SYSTEM CODEC_TEST2L (* PUBL/SUBL Test with Derived Data Types *)
  (* Standard: 61499-1ITA; Classification: Communications; Function: Test System *)
  (* Version 0.9, 2004-06-23, JHC, Rockwell Automation, Deleted MONITOR (not used). *)
  (* Version 0.8, 2004-06-22, JHC, Rockwell Automation, Modified to use IN_MATRIX, OUT_MATRIX. *)
  (* Version 0.7, 2003-12-04, JHC, Rockwell Automation, Removed QI's from PUBL/SUBLs *)
  (* Version 0.6, 2002-03-08, JHC, Rockwell Automation, Added M_IO for MATRIX I/O *)
  (* Version 0.5, 2002-03-06, JHC, Rockwell Automation, Added TEST_MATRIX, single TEST frame *)
  (* Version 0.4, 2001-06-13, JHC, Rockwell Automation, Added applications including TEST_AI16C. *)
  (* Version 0.3, 2001-06-08, JHC, Rockwell Automation, Corrected UDP addresses; changed GUIs to IN_ANY, OUT_ANY *)
  (* Version 0.2, 2001-05-30, JHC, Rockwell Automation, Saved layouts *)
  (* Version 0.1, 2000-05-16, JHC, Rockwell Automation, File type changed to ".sys" *)
  (* Version 0.0, 2000-04-19, JHC, Rockwell Automation *)
  APPLICATION TEST_REAL_VS
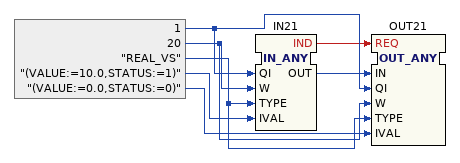
    FBS
      IN21 : IN_ANY;
      OUT21 : OUT_ANY;
    END_FBS
    EVENT_CONNECTIONS
      IN21.IND TO OUT21.REQ;
    END_CONNECTIONS
    DATA_CONNECTIONS
      IN21.OUT TO OUT21.IN;
      1 TO IN21.QI;
      20 TO IN21.W;
      "REAL_VS" TO IN21.TYPE;
      "(VALUE:=10.0,STATUS:=1)" TO IN21.IVAL;
      1 TO OUT21.QI;
      20 TO OUT21.W;
      "REAL_VS" TO OUT21.TYPE;
      "(VALUE:=0.0,STATUS:=0)" TO OUT21.IVAL;
    END_CONNECTIONS
  END_APPLICATION
  APPLICATION TEST_ENUMS
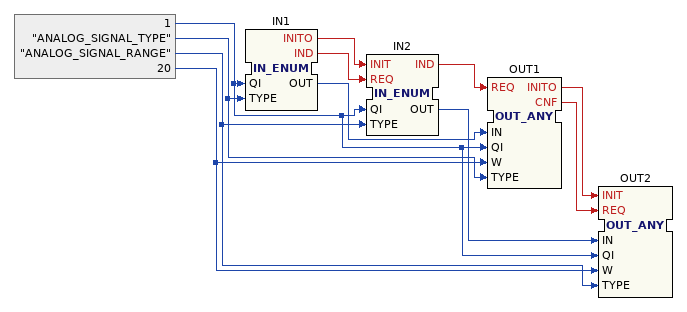
    FBS
      IN1 : IN_ENUM;
      IN2 : IN_ENUM;
      OUT1 : OUT_ANY;
      OUT2 : OUT_ANY;
    END_FBS
    EVENT_CONNECTIONS
      IN1.INITO TO IN2.INIT;
      IN1.IND TO IN2.REQ;
      IN2.IND TO OUT1.REQ;
      OUT1.INITO TO OUT2.INIT;
      OUT1.CNF TO OUT2.REQ;
    END_CONNECTIONS
    DATA_CONNECTIONS
      IN1.OUT TO OUT1.IN;
      IN2.OUT TO OUT2.IN;
      1 TO IN1.QI;
      "ANALOG_SIGNAL_TYPE" TO IN1.TYPE;
      1 TO IN2.QI;
      "ANALOG_SIGNAL_RANGE" TO IN2.TYPE;
      1 TO OUT1.QI;
      20 TO OUT1.W;
      "ANALOG_SIGNAL_TYPE" TO OUT1.TYPE;
      1 TO OUT2.QI;
      20 TO OUT2.W;
      "ANALOG_SIGNAL_RANGE" TO OUT2.TYPE;
    END_CONNECTIONS
  END_APPLICATION
  APPLICATION TEST_FREQ
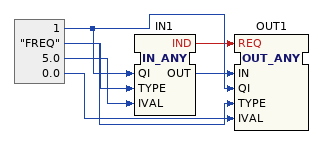
    FBS
      IN1 : IN_ANY;
      OUT1 : OUT_ANY;
    END_FBS
    EVENT_CONNECTIONS
      IN1.IND TO OUT1.REQ;
    END_CONNECTIONS
    DATA_CONNECTIONS
      IN1.OUT TO OUT1.IN;
      1 TO IN1.QI;
      "FREQ" TO IN1.TYPE;
      5.0 TO IN1.IVAL;
      1 TO OUT1.QI;
      "FREQ" TO OUT1.TYPE;
      0.0 TO OUT1.IVAL;
    END_CONNECTIONS
  END_APPLICATION
  APPLICATION TEST_SUBR
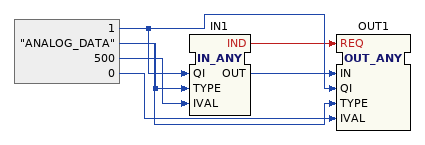
    FBS
      IN1 : IN_ANY;
      OUT1 : OUT_ANY;
    END_FBS
    EVENT_CONNECTIONS
      IN1.IND TO OUT1.REQ;
    END_CONNECTIONS
    DATA_CONNECTIONS
      IN1.OUT TO OUT1.IN;
      1 TO IN1.QI;
      "ANALOG_DATA" TO IN1.TYPE;
      500 TO IN1.IVAL;
      1 TO OUT1.QI;
      "ANALOG_DATA" TO OUT1.TYPE;
      0 TO OUT1.IVAL;
    END_CONNECTIONS
  END_APPLICATION
  APPLICATION TEST_AI16
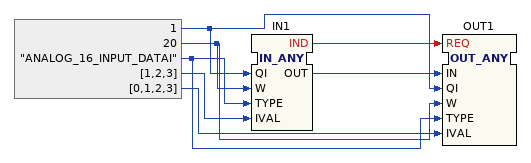
    FBS
      IN1 : IN_ANY;
      OUT1 : OUT_ANY;
    END_FBS
    EVENT_CONNECTIONS
      IN1.IND TO OUT1.REQ;
    END_CONNECTIONS
    DATA_CONNECTIONS
      IN1.OUT TO OUT1.IN;
      1 TO IN1.QI;
      20 TO IN1.W;
      "ANALOG_16_INPUT_DATAI" TO IN1.TYPE;
      [1,2,3] TO IN1.IVAL;
      1 TO OUT1.QI;
      20 TO OUT1.W;
      "ANALOG_16_INPUT_DATAI" TO OUT1.TYPE;
      [0,1,2,3] TO OUT1.IVAL;
    END_CONNECTIONS
  END_APPLICATION
  APPLICATION TEST_AI16C (* Test ANALOG_16_INPUT_CONFIGURATION *)
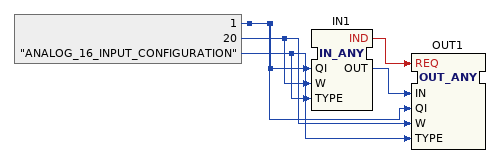
    FBS
      IN1 : IN_ANY;
      OUT1 : OUT_ANY;
    END_FBS
    EVENT_CONNECTIONS
      IN1.IND TO OUT1.REQ;
    END_CONNECTIONS
    DATA_CONNECTIONS
      IN1.OUT TO OUT1.IN;
      1 TO IN1.QI;
      1 TO OUT1.QI;
      20 TO IN1.W;
      "ANALOG_16_INPUT_CONFIGURATION" TO IN1.TYPE;
      20 TO OUT1.W;
      "ANALOG_16_INPUT_CONFIGURATION" TO OUT1.TYPE;
    END_CONNECTIONS
  END_APPLICATION
  APPLICATION TEST_MATRIX
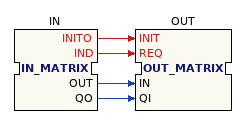
    FBS
      IN : IN_MATRIX;
      OUT : OUT_MATRIX;
    END_FBS
    EVENT_CONNECTIONS
      IN.INITO TO OUT.INIT;
      IN.IND TO OUT.REQ;
    END_CONNECTIONS
    DATA_CONNECTIONS
      IN.OUT TO OUT.IN;
      IN.QO TO OUT.QI;
    END_CONNECTIONS
  END_APPLICATION
  DEVICE TEST : FRAME_DEVICE
    RESOURCE SEND_REAL_VS : PANEL_RESOURCE
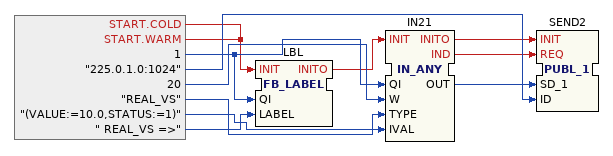
      FBS
        LBL : FB_LABEL;
        IN21 : IN_ANY;
        SEND2 : PUBL_1;
      END_FBS
      EVENT_CONNECTIONS
        START.COLD TO LBL.INIT;
        START.WARM TO LBL.INIT;
        LBL.INITO TO IN21.INIT;
        IN21.INITO TO SEND2.INIT;
        IN21.IND TO SEND2.REQ;
      END_CONNECTIONS
      DATA_CONNECTIONS
        1 TO IN21.QI;
        IN21.OUT TO SEND2.SD_1;
        "225.0.1.0:1024" TO SEND2.ID;
        20 TO IN21.W;
        "REAL_VS" TO IN21.TYPE;
        "(VALUE:=10.0,STATUS:=1)" TO IN21.IVAL;
        1 TO LBL.QI;
        " REAL_VS =>" TO LBL.LABEL;
      END_CONNECTIONS
    END_RESOURCE
    RESOURCE RCV_REAL_VS : PANEL_RESOURCE
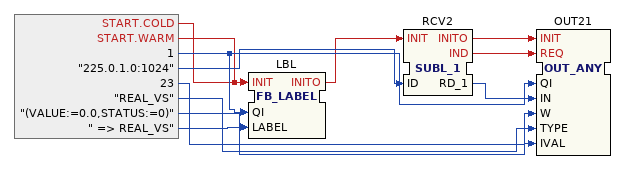
      FBS
        LBL : FB_LABEL;
        RCV2 : SUBL_1;
        OUT21 : OUT_ANY;
      END_FBS
      EVENT_CONNECTIONS
        START.COLD TO LBL.INIT;
        START.WARM TO LBL.INIT;
        LBL.INITO TO RCV2.INIT;
        RCV2.INITO TO OUT21.INIT;
        RCV2.IND TO OUT21.REQ;
      END_CONNECTIONS
      DATA_CONNECTIONS
        1 TO OUT21.QI;
        RCV2.RD_1 TO OUT21.IN;
        "225.0.1.0:1024" TO RCV2.ID;
        23 TO OUT21.W;
        "REAL_VS" TO OUT21.TYPE;
        "(VALUE:=0.0,STATUS:=0)" TO OUT21.IVAL;
        1 TO LBL.QI;
        " => REAL_VS" TO LBL.LABEL;
      END_CONNECTIONS
    END_RESOURCE
    RESOURCE SEND_ENUMS : PANEL_RESOURCE
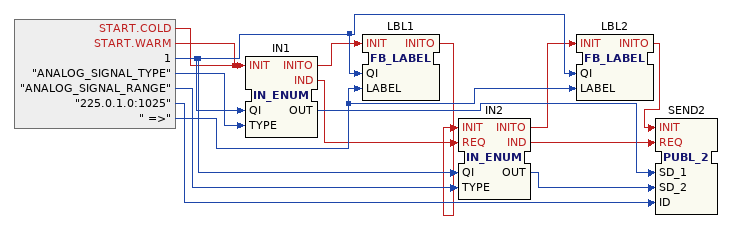
      FBS
        IN1 : IN_ENUM;
        LBL1 : FB_LABEL;
        IN2 : IN_ENUM;
        LBL2 : FB_LABEL;
        SEND2 : PUBL_2;
      END_FBS
      EVENT_CONNECTIONS
        START.COLD TO IN1.INIT;
        START.WARM TO IN1.INIT;
        IN1.INITO TO LBL1.INIT;
        LBL1.INITO TO IN2.INIT;
        IN2.INITO TO LBL2.INIT;
        LBL2.INITO TO SEND2.INIT;
        IN1.IND TO IN2.REQ;
        IN2.IND TO SEND2.REQ;
      END_CONNECTIONS
      DATA_CONNECTIONS
        1 TO IN1.QI;
        1 TO IN2.QI;
        IN1.OUT TO SEND2.SD_1;
        IN2.OUT TO SEND2.SD_2;
        "ANALOG_SIGNAL_TYPE" TO IN1.TYPE;
        "ANALOG_SIGNAL_RANGE" TO IN2.TYPE;
        "225.0.1.0:1025" TO SEND2.ID;
        1 TO LBL1.QI;
        " =>" TO LBL1.LABEL;
        1 TO LBL2.QI;
        " =>" TO LBL2.LABEL;
      END_CONNECTIONS
    END_RESOURCE
    RESOURCE RCV_ENUMS : PANEL_RESOURCE
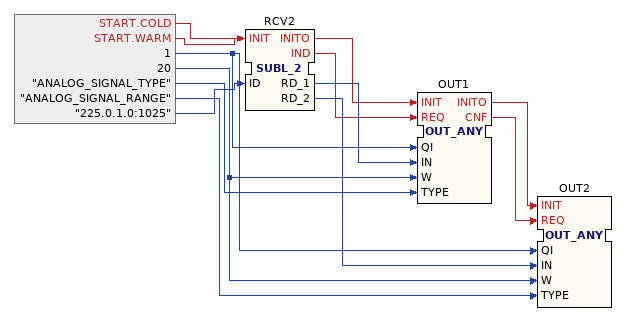
      FBS
        RCV2 : SUBL_2;
        OUT1 : OUT_ANY;
        OUT2 : OUT_ANY;
      END_FBS
      EVENT_CONNECTIONS
        START.COLD TO RCV2.INIT;
        START.WARM TO RCV2.INIT;
        RCV2.INITO TO OUT1.INIT;
        OUT1.INITO TO OUT2.INIT;
        RCV2.IND TO OUT1.REQ;
        OUT1.CNF TO OUT2.REQ;
      END_CONNECTIONS
      DATA_CONNECTIONS
        1 TO OUT1.QI;
        1 TO OUT2.QI;
        RCV2.RD_1 TO OUT1.IN;
        RCV2.RD_2 TO OUT2.IN;
        20 TO OUT1.W;
        "ANALOG_SIGNAL_TYPE" TO OUT1.TYPE;
        20 TO OUT2.W;
        "ANALOG_SIGNAL_RANGE" TO OUT2.TYPE;
        "225.0.1.0:1025" TO RCV2.ID;
      END_CONNECTIONS
    END_RESOURCE
    RESOURCE SEND_FREQ : PANEL_RESOURCE
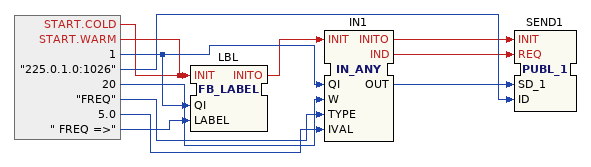
      FBS
        LBL : FB_LABEL;
        IN1 : IN_ANY;
        SEND1 : PUBL_1;
      END_FBS
      EVENT_CONNECTIONS
        START.COLD TO LBL.INIT;
        START.WARM TO LBL.INIT;
        LBL.INITO TO IN1.INIT;
        IN1.INITO TO SEND1.INIT;
        IN1.IND TO SEND1.REQ;
      END_CONNECTIONS
      DATA_CONNECTIONS
        1 TO IN1.QI;
        IN1.OUT TO SEND1.SD_1;
        "225.0.1.0:1026" TO SEND1.ID;
        20 TO IN1.W;
        "FREQ" TO IN1.TYPE;
        5.0 TO IN1.IVAL;
        1 TO LBL.QI;
        " FREQ =>" TO LBL.LABEL;
      END_CONNECTIONS
    END_RESOURCE
    RESOURCE RCV_FREQ : PANEL_RESOURCE
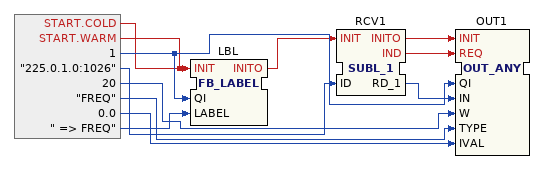
      FBS
        LBL : FB_LABEL;
        RCV1 : SUBL_1;
        OUT1 : OUT_ANY;
      END_FBS
      EVENT_CONNECTIONS
        START.COLD TO LBL.INIT;
        START.WARM TO LBL.INIT;
        LBL.INITO TO RCV1.INIT;
        RCV1.INITO TO OUT1.INIT;
        RCV1.IND TO OUT1.REQ;
      END_CONNECTIONS
      DATA_CONNECTIONS
        1 TO OUT1.QI;
        RCV1.RD_1 TO OUT1.IN;
        "225.0.1.0:1026" TO RCV1.ID;
        20 TO OUT1.W;
        "FREQ" TO OUT1.TYPE;
        0.0 TO OUT1.IVAL;
        1 TO LBL.QI;
        " => FREQ" TO LBL.LABEL;
      END_CONNECTIONS
    END_RESOURCE
    RESOURCE SEND_SUBR : PANEL_RESOURCE
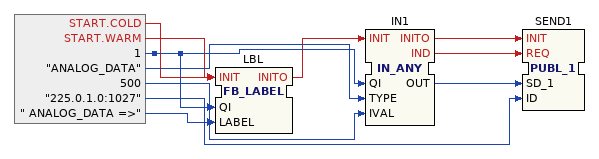
      FBS
        LBL : FB_LABEL;
        IN1 : IN_ANY;
        SEND1 : PUBL_1;
      END_FBS
      EVENT_CONNECTIONS
        START.COLD TO LBL.INIT;
        START.WARM TO LBL.INIT;
        LBL.INITO TO IN1.INIT;
        IN1.INITO TO SEND1.INIT;
        IN1.IND TO SEND1.REQ;
      END_CONNECTIONS
      DATA_CONNECTIONS
        1 TO IN1.QI;
        IN1.OUT TO SEND1.SD_1;
        "ANALOG_DATA" TO IN1.TYPE;
        500 TO IN1.IVAL;
        "225.0.1.0:1027" TO SEND1.ID;
        1 TO LBL.QI;
        " ANALOG_DATA =>" TO LBL.LABEL;
      END_CONNECTIONS
    END_RESOURCE
    RESOURCE RCV_SUBR : PANEL_RESOURCE
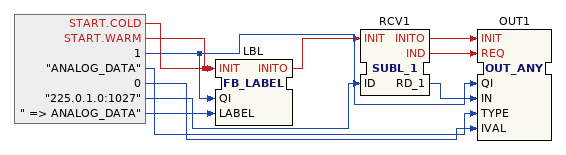
      FBS
        LBL : FB_LABEL;
        RCV1 : SUBL_1;
        OUT1 : OUT_ANY;
      END_FBS
      EVENT_CONNECTIONS
        START.COLD TO LBL.INIT;
        START.WARM TO LBL.INIT;
        LBL.INITO TO RCV1.INIT;
        RCV1.INITO TO OUT1.INIT;
        RCV1.IND TO OUT1.REQ;
      END_CONNECTIONS
      DATA_CONNECTIONS
        1 TO OUT1.QI;
        RCV1.RD_1 TO OUT1.IN;
        "ANALOG_DATA" TO OUT1.TYPE;
        0 TO OUT1.IVAL;
        "225.0.1.0:1027" TO RCV1.ID;
        1 TO LBL.QI;
        " => ANALOG_DATA" TO LBL.LABEL;
      END_CONNECTIONS
    END_RESOURCE
    RESOURCE SEND_AI16 : PANEL_RESOURCE
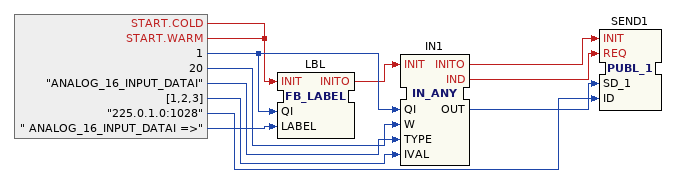
      FBS
        LBL : FB_LABEL;
        IN1 : IN_ANY;
        SEND1 : PUBL_1;
      END_FBS
      EVENT_CONNECTIONS
        START.COLD TO LBL.INIT;
        START.WARM TO LBL.INIT;
        LBL.INITO TO IN1.INIT;
        IN1.INITO TO SEND1.INIT;
        IN1.IND TO SEND1.REQ;
      END_CONNECTIONS
      DATA_CONNECTIONS
        1 TO IN1.QI;
        IN1.OUT TO SEND1.SD_1;
        20 TO IN1.W;
        "ANALOG_16_INPUT_DATAI" TO IN1.TYPE;
        [1,2,3] TO IN1.IVAL;
        "225.0.1.0:1028" TO SEND1.ID;
        1 TO LBL.QI;
        " ANALOG_16_INPUT_DATAI =>" TO LBL.LABEL;
      END_CONNECTIONS
    END_RESOURCE
    RESOURCE RCV_AI16 : PANEL_RESOURCE
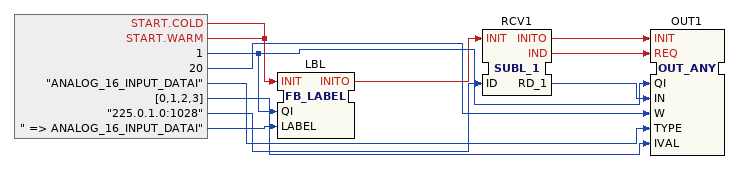
      FBS
        LBL : FB_LABEL;
        RCV1 : SUBL_1;
        OUT1 : OUT_ANY;
      END_FBS
      EVENT_CONNECTIONS
        START.COLD TO LBL.INIT;
        START.WARM TO LBL.INIT;
        LBL.INITO TO RCV1.INIT;
        RCV1.INITO TO OUT1.INIT;
        RCV1.IND TO OUT1.REQ;
      END_CONNECTIONS
      DATA_CONNECTIONS
        1 TO OUT1.QI;
        RCV1.RD_1 TO OUT1.IN;
        20 TO OUT1.W;
        "ANALOG_16_INPUT_DATAI" TO OUT1.TYPE;
        [0,1,2,3] TO OUT1.IVAL;
        "225.0.1.0:1028" TO RCV1.ID;
        1 TO LBL.QI;
        " => ANALOG_16_INPUT_DATAI" TO LBL.LABEL;
      END_CONNECTIONS
    END_RESOURCE
    RESOURCE SEND_AI16C : PANEL_RESOURCE
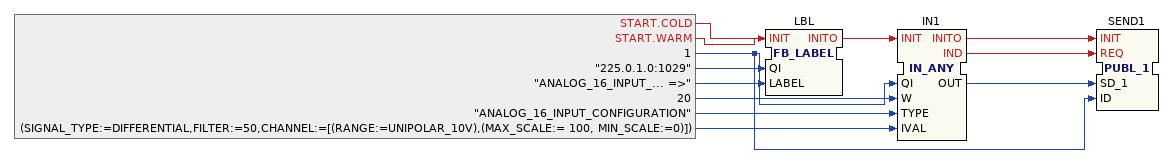
      FBS
        LBL : FB_LABEL;
        IN1 : IN_ANY;
        SEND1 : PUBL_1;
      END_FBS
      EVENT_CONNECTIONS
        START.COLD TO LBL.INIT;
        START.WARM TO LBL.INIT;
        LBL.INITO TO IN1.INIT;
        IN1.INITO TO SEND1.INIT;
        IN1.IND TO SEND1.REQ;
      END_CONNECTIONS
      DATA_CONNECTIONS
        IN1.OUT TO SEND1.SD_1;
        1 TO IN1.QI;
        "225.0.1.0:1029" TO SEND1.ID;
        1 TO LBL.QI;
        "ANALOG_16_INPUT_... =>" TO LBL.LABEL;
        20 TO IN1.W;
        "ANALOG_16_INPUT_CONFIGURATION" TO IN1.TYPE;
        (SIGNAL_TYPE:=DIFFERENTIAL,FILTER:=50,CHANNEL:=[(RANGE:=UNIPOLAR_10V),(MAX_SCALE:= 100, MIN_SCALE:=0)]) TO IN1.IVAL;
      END_CONNECTIONS
    END_RESOURCE
    RESOURCE RCV_AI16C : PANEL_RESOURCE
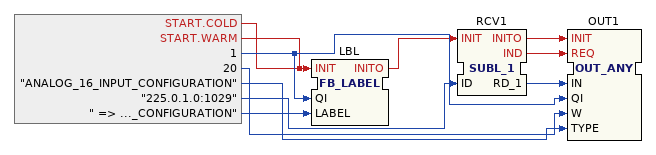
      FBS
        LBL : FB_LABEL;
        RCV1 : SUBL_1;
        OUT1 : OUT_ANY;
      END_FBS
      EVENT_CONNECTIONS
        START.COLD TO LBL.INIT;
        START.WARM TO LBL.INIT;
        LBL.INITO TO RCV1.INIT;
        RCV1.INITO TO OUT1.INIT;
        RCV1.IND TO OUT1.REQ;
      END_CONNECTIONS
      DATA_CONNECTIONS
        RCV1.RD_1 TO OUT1.IN;
        1 TO OUT1.QI;
        20 TO OUT1.W;
        "ANALOG_16_INPUT_CONFIGURATION" TO OUT1.TYPE;
        "225.0.1.0:1029" TO RCV1.ID;
        1 TO LBL.QI;
        " => ..._CONFIGURATION" TO LBL.LABEL;
      END_CONNECTIONS
    END_RESOURCE
    RESOURCE SEND_MATRIX : PANEL_RESOURCE
      FBS
        IN1 : IN_MATRIX;
        SEND1 : PUBL_1;
      END_FBS
      EVENT_CONNECTIONS
        START.COLD TO IN1.INIT;
        START.WARM TO IN1.INIT;
        IN1.IND TO SEND1.REQ;
        IN1.INITO TO SEND1.INIT;
      END_CONNECTIONS
      DATA_CONNECTIONS
        IN1.OUT TO SEND1.SD_1;
        1 TO IN1.QI;
        "225.0.1.0:1030" TO SEND1.ID;
        2 TO IN1.ROWS;
        3 TO IN1.COLS;
        [1,2,3,4,5,6] TO IN1.IVAL;
      END_CONNECTIONS
    END_RESOURCE
    RESOURCE RCV_MATRIX : PANEL_RESOURCE
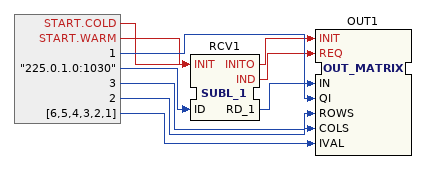
      FBS
        RCV1 : SUBL_1;
        OUT1 : OUT_MATRIX;
      END_FBS
      EVENT_CONNECTIONS
        START.COLD TO RCV1.INIT;
        START.WARM TO RCV1.INIT;
        RCV1.INITO TO OUT1.INIT;
        RCV1.IND TO OUT1.REQ;
      END_CONNECTIONS
      DATA_CONNECTIONS
        RCV1.RD_1 TO OUT1.IN;
        1 TO OUT1.QI;
        "225.0.1.0:1030" TO RCV1.ID;
        3 TO OUT1.ROWS;
        2 TO OUT1.COLS;
        [6,5,4,3,2,1] TO OUT1.IVAL;
      END_CONNECTIONS
    END_RESOURCE
    DATA_CONNECTIONS
      1 TO SEND_MATRIX.ROWS;
      1 TO SEND_MATRIX.COLS;
      1 TO RCV_MATRIX.ROWS;
      1 TO RCV_MATRIX.COLS;
    END_CONNECTIONS
  END_DEVICE
  DATA_CONNECTIONS (* parameter values *)
    [100,250,800,320] TO TEST.BOUNDS;
    [4,4] TO TEST.GRID;
  END_CONNECTIONS
END_SYSTEM
